Staubli VAL3: ReadSingTraj.pgx

public program ReadSingTraj(string x_sTrajName, bool& x_bRes)
  local num l_nNum[3]
  local num l_nTrajIndex
  local string l_sBuff
  local string l_sFileName
  local trsf l_trTrsf
begin

  //读取生产文件
  //生产文件格式按照LasMAN3.7格式进行


  //参数初始化
  x_bRes=false
  l_sFileName="Disk://Txt/Traj.txt"

  //判断文件是否存在
  if !$fileExists(l_sFileName)
    return
  endIf

  //关闭所有文件
  call FileDir:CloseAllFile()

  //文件是否可以打开
  nFileID=$fileOpen(l_sFileName,"r")
  if nFileID<0 or nFileID>9
    return
  endIf



  //读取每行并解析
  if $fileGet(nFileID,l_sBuff,1)!=1 or find(l_sBuff,"BEGIN="+x_sTrajName)<0
    return
  endIf

  if $fileGet(nFileID,l_sBuff,1)!=1 or find(l_sBuff,"BYPASS=")<0
    return
  endIf

  call ReadPoint(x_bRes)
  //关闭所有文件
  call FileDir:CloseAllFile()
end
